(*Vincent Molenkamp : 519540*)
FUNCTION ScaleOutput : DINT
(*Om de output waarde te scalen naar Van DINT naar WORD*)
VAR_INPUT	
	Input: INT;	  (*waarde die gescaled moet worden*)
	Minimum: INT; (*De minimum input waarde*)
	Maximum: INT; (*De maximum input waarde*)
END_VAR
VAR
	X: DINT;
END_VAR

(* To set minimum and maximum values for the input *)
IF Input < Minimum THEN
	Input := Minimum;
ELSIF Input > Maximum THEN
	Input := Maximum;
END_IF

(* Calculating the output value does not work with negative minimum *) 
ScaleOutput := ((Input-Minimum)*65535)/(Maximum-Minimum);

END_FUNCTION

(* stored: Version 1.1.0.1, ProductVersion 3.1.4024.12
   POU ScaleOutput: Id {3c790d3f-23db-4dd3-a7f4-8c78888ec7ed}, SpecialFunc None *)
